FUNCTION_BLOCK FB_PowerAll
VAR_INPUT
	Enable 		: BOOL;
END_VAR
VAR_OUTPUT
	Status		: BOOL;
	Error		: BOOL;
	Done		: BOOL;
END_VAR
VAR
	fbPower 		: ARRAY [1..GVL_XY.cAxesCount] OF MC_Power;
	i				: UINT;
	fbPowerSlave 	: ARRAY [1..GVL_XY.cAxesSlaveCount] OF MC_Power;
END_VAR

IF Enable THEN
	Status := TRUE;
	Error := FALSE;
	Done := FALSE;
	
	FOR i:=1 TO GVL_XY.cAxesCount DO
		fbPower[i](Axis:=GVL_XY.stAxis[i],
			Enable			:= Enable,
			Enable_Positive	:= Enable,
			Enable_Negative	:= Enable
		);
		
		Status := Status AND fbPower[i].Status; 
		Error := Error OR fbPower[i].Error;
	END_FOR
	
	FOR i:= 1 TO GVL_XY.cAxesSlaveCount DO
		fbPowerSlave[i](
			Axis := GVL_XY.stSlaveAxis[i],
			Enable			:= Enable,
			Enable_Positive	:= Enable,
			Enable_Negative	:= Enable	
			);
			
		Status := Status AND fbPowerSlave[i].Status; 
		Error := Error OR fbPowerSlave[i].Error;
	END_FOR
	
	IF Status AND NOT Error THEN
		Done := TRUE;
	END_IF
END_IF

END_FUNCTION_BLOCK

(* stored: Version 1.1.0.1, ProductVersion 3.1.4024.11
   POU FB_PowerAll: Id {d3e6d2d4-b215-4a84-8022-bf06b4a82234}, SpecialFunc None *)
